PROGRAM Motor_move
VAR
	motorDirection_rotate: Motor_Direction;
	position_rotation: UINT;
	writeRotateReference: BOOL;
	writeHorizontalReference: BOOL;
	writeVerticalReference: BOOL;
	tolerance: UINT :=20;
	movemotor_rotate: Motor_Enable;
	desiredSpeed: INT :=5000;
END_VAR

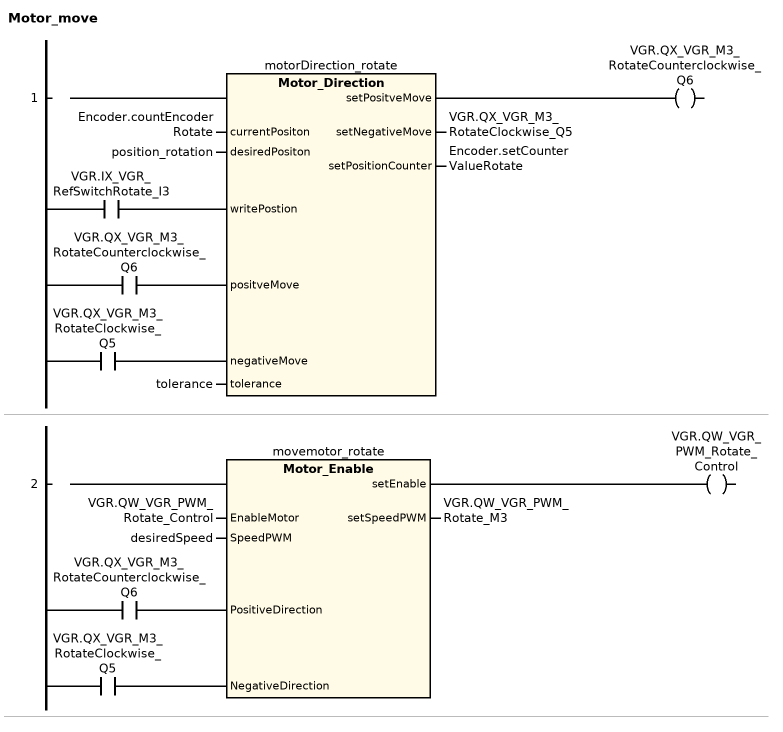
// NETWORK 1
motorDirection_rotate(
    currentPositon := Encoder.countEncoderRotate,
    desiredPositon := position_rotation,
    writePostion := VGR.IX_VGR_RefSwitchRotate_I3,
    positveMove := VGR.QX_VGR_M3_RotateCounterclockwise_Q6,
    negativeMove := VGR.QX_VGR_M3_RotateClockwise_Q5,
    tolerance := tolerance,
    setNegativeMove => VGR.QX_VGR_M3_RotateClockwise_Q5,
    setPositionCounter => Encoder.setCounterValueRotate); // Motor_Direction
VGR.QX_VGR_M3_RotateCounterclockwise_Q6 := motorDirection_rotate.setPositveMove;

// NETWORK 2
movemotor_rotate(
    EnableMotor := VGR.QW_VGR_PWM_Rotate_Control,
    SpeedPWM := desiredSpeed,
    PositiveDirection := VGR.QX_VGR_M3_RotateCounterclockwise_Q6,
    NegativeDirection := VGR.QX_VGR_M3_RotateClockwise_Q5,
    setSpeedPWM => VGR.QW_VGR_PWM_Rotate_M3); // Motor_Enable
VGR.QW_VGR_PWM_Rotate_Control := movemotor_rotate.setEnable;

END_PROGRAM

(* stored: Version 1.1.0.1, ProductVersion 3.1.4024.12
   POU Motor_move: Id {9a04db00-abe5-4125-8ad3-35cb329d63fd}, SpecialFunc None *)
